TYPE ST_BaseRecipe_HMI :
STRUCT
END_STRUCT
END_TYPE

(* stored: Version 1.1.0.1
   DUT ST_BaseRecipe_HMI: Id {bcd1daa3-b028-01ce-1df0-56bbd28ee1cb} *)
